# B&R Automation Studio project StructureSample
Automation Studio 4.12.8.41 SP

## Configuration Config1

CPU PC_any, AutomationRuntime Q4.93, Build 4.1.2, Vc V4.73.3

### Task classes (Cpu.sw)
```
Cyclic#8 (cycle 50000 us):
  StructureT <- GetVarStructure.prg
Binaries: udbdef, FWRules, TCData, iomap, ashwac, Role, sysconf, arconfig, asfw, User, ashwd
Libraries: AsBrStr, sys_lib, ArEventLog, runtime, AdvIecChk
```

### Hardware
```
PC : PC_any v1.1.1.0 (OrderNumber=PC)
  ConfigurationID = StructureTest_Config1
  Cyclic8Duration = 50000
  FileDevice1
  FileDeviceName1 = USER
  FileDevicePath1 = USER_PATH
```

## Logical view

Binary libraries used (declarations not repeated): operator, runtime, astime, AsIecCon, AsBrStr, sys_lib, ArEventLog

### Global.typ - Global data types
```iecst
TYPE
	testEnum :
		(
		red,
		green
		);
	testStructure : 	STRUCT
		Var1 : USINT;
		Var2 : UDINT;
		Var3 : ARRAY[0..5]OF UDINT;
		Enum : testEnum;
		RealLongVariableName : testSubStructure;
		SubStructure : testSubSubStructure;
	END_STRUCT;
	testSubStructure : 	STRUCT
		Var1234567 : STRING[80];
		Var22 : UDINT;
		EvenLongerSubVariableName : testSubSubStructure;
	END_STRUCT;
	testSubSubStructure : 	STRUCT
		Var11 : STRING[80];
		Var22 : UDINT;
		TheLongestSubVariableNameInisde : ARRAY[0..5]OF USINT;
	END_STRUCT;
END_TYPE
```

### Global.var - Global variables
```iecst
VAR
	testvariable_org : testStructure;
	testvariable_cpy : testStructure;
END_VAR
```

### Package Logical/Libraries - Global libraries

### Library Logical/Libraries/AdvIecChk (IEC, version 2.00.0) - IEC Check w/ Advanced Debugging Data
Depends on: Sys_Lib, AsBrStr, ArEventLog

#### AdvIecChk.fun - Exported functions and function blocks
```iecst
(************************************************************************************

Advanced IEC Check Functions Library

File: AdvIecChk.fun
Description: Declaration of library functions

!! Note: See the Automation Studio Help file before modifying these declarations!   !!
!! Most of these functions must be declared exactly as-is in order for the          !!
!! processor to recognize them as check functions. The implementation can change    !!
!! but the declaration cannot!                                                      !!

Authors:
    - Matt Adams (B&R Industrial Automation)
    - Varad Darji (B&R Industrial Automation)
    - Marcus Mangel (B&R Industrial Automation)

************************************************************************************)

FUNCTION CheckDivSint : SINT (*Called before the division/module using a SINT value. Returns the divisor if no errors are found*)
	VAR_INPUT
		divisor : SINT; (*For division: Value that should be divided by. For modulo: Right operand*)
	END_VAR
END_FUNCTION

FUNCTION CheckDivUsint : USINT (*Called before the division/module using a USINT value. Returns the divisor if no errors are found*)
	VAR_INPUT
		divisor : USINT; (*For division: Value that should be divided by. For modulo: Right operand*)
	END_VAR
END_FUNCTION

FUNCTION CheckDivInt : INT (*Called before the division/module using a INT value. Returns the divisor if no errors are found*)
	VAR_INPUT
		divisor : INT; (*For division: Value that should be divided by. For modulo: Right operand*)
	END_VAR
END_FUNCTION

FUNCTION CheckDivUint : UINT (*Called before the division/module using a UINT value. Returns the divisor if no errors are found*)
	VAR_INPUT
		divisor : UINT; (*For division: Value that should be divided by. For modulo: Right operand*)
	END_VAR
END_FUNCTION

FUNCTION CheckDivDint : DINT (*Called before the division/module using a DINT value. Returns the divisor if no errors are found*)
	VAR_INPUT
		divisor : DINT; (*For division: Value that should be divided by. For modulo: Right operand*)
	END_VAR
END_FUNCTION

FUNCTION CheckDivUdint : UDINT (*Called before the division/module using a UDINT value. Returns the divisor if no errors are found*)
	VAR_INPUT
		divisor : UDINT; (*For division: Value that should be divided by. For modulo: Right operand*)
	END_VAR
END_FUNCTION

FUNCTION CheckDivReal : REAL (*Called before the division/module using a REAL value. Returns the divisor if no errors are found*)
	VAR_INPUT
		divisor : REAL; (*For division: Value that should be divided by. For modulo: Right operand*)
	END_VAR
END_FUNCTION

FUNCTION CheckDivLReal : LREAL (*Called before the division/module using a LREAL value. Returns the divisor if no errors are found. (Cannot be used on SG3 or SGC targets)*)
	VAR_INPUT
		divisor : LREAL; (*For division: Value that should be divided by. For modulo: Right operand*)
	END_VAR
END_FUNCTION

FUNCTION CheckBounds : DINT (*Called before accessing an array. Returns the index if no errors are found. Otherwise, returns the problematic index bound*)
	VAR_INPUT
		index : DINT; (*Index being accessed*)
		lower : DINT; (*Lower bound (lowest possible index) of the array*)
		upper : DINT; (*Upper bound (highest possible index) of the array*)
	END_VAR
	VAR
		LowString : STRING[ADVIECCHK_MAX_STRING_LEN]; (*[INTERNAL] Lower bound as a string*)
		UpString : STRING[ADVIECCHK_MAX_STRING_LEN]; (*[INTERNAL] Upper bound as a string*)
		IndexString : STRING[ADVIECCHK_MAX_STRING_LEN]; (*[INTERNAL] Index as a string*)
		ErrorText : STRING[ADVIECCHK_MAX_STRING_LEN]; (*[INTERNAL] Error text created for a long entry based on input data*)
	END_VAR
END_FUNCTION

FUNCTION CheckRange : DINT (*Called before write accessing an enumeration variable. Returns the value if no errors are found. Otherwise, returns the problematic value bound*)
	VAR_INPUT
		value : DINT; (*Enumeration value being accessed*)
		lower : DINT; (*Lower bound (lowest possible value) of the enumeration*)
		upper : DINT; (*Upper bound (highest possible value) of the enumeration*)
	END_VAR
	VAR
		LowString : STRING[ADVIECCHK_MAX_STRING_LEN]; (*[INTERNAL] Lower bound as a string*)
		UpString : STRING[ADVIECCHK_MAX_STRING_LEN]; (*[INTERNAL] Upper bound as a string*)
		ValueString : STRING[ADVIECCHK_MAX_STRING_LEN]; (*[INTERNAL] Value as a string*)
		ErrorText : STRING[ADVIECCHK_MAX_STRING_LEN]; (*[INTERNAL] Error text created for a long entry based on input data*)
	END_VAR
END_FUNCTION

FUNCTION CheckSignedSubrange : DINT (*Called before write access to a variable with the data type "Subrange" if the subrange is used on a signed data type. Returns the value if no errors are found.
Otherwise, returns the problematic value bound*)
	VAR_INPUT
		value : DINT; (*Index being accessed*)
		lower : DINT; (*Lower bound (lowest possible index) of the subrange*)
		upper : DINT; (*Upper bound (highest possible index) of the subrange*)
	END_VAR
	VAR
		LowString : STRING[ADVIECCHK_MAX_STRING_LEN]; (*[INTERNAL] Lower bound as a string*)
		UpString : STRING[ADVIECCHK_MAX_STRING_LEN]; (*[INTERNAL] Lower bound as a string*)
		ValueString : STRING[ADVIECCHK_MAX_STRING_LEN]; (*[INTERNAL] Value as a string*)
		ErrorText : STRING[ADVIECCHK_MAX_STRING_LEN]; (*[INTERNAL] Error text created for a long entry based on input data*)
	END_VAR
END_FUNCTION

FUNCTION CheckUnsignedSubrange : UDINT (*Called before write access to a variable with the data type "Subrange" if the subrange is used on an unsigned data type. Returns the value if no errors are found.
Otherwise, returns the problematic value bound*)
	VAR_INPUT
		value : UDINT; (*Index being accessed*)
		lower : UDINT; (*Lower bound (lowest possible index) of the subrange*)
		upper : UDINT; (*Upper bound (highest possible index) of the subrange*)
	END_VAR
	VAR
		LowString : STRING[ADVIECCHK_MAX_STRING_LEN]; (*[INTERNAL] Lower bound as a string*)
		UpString : STRING[ADVIECCHK_MAX_STRING_LEN]; (*[INTERNAL] Upper bound as a string*)
		ValueString : STRING[ADVIECCHK_MAX_STRING_LEN]; (*[INTERNAL] Value as a string*)
		ErrorText : STRING[ADVIECCHK_MAX_STRING_LEN]; (*[INTERNAL] Error text created for a long entry based on input data*)
	END_VAR
END_FUNCTION

FUNCTION CheckReadAccess : UDINT (*Called before (read) accessing a memory address using a dynamic variable (ADR). Returns the input address*)
	VAR_INPUT
		address : UDINT; (*Address of the memory area being accessed*)
	END_VAR
END_FUNCTION

FUNCTION CheckWriteAccess : UDINT (*Called before (write) accessing a memory address using a dynamic variable (ADR). Returns the input address*)
	VAR_INPUT
		address : UDINT; (*Address of the memory area being accessed*)
	END_VAR
END_FUNCTION

FUNCTION MakeEntry : UDINT (*Creates a Logger entry detailing any errors. Returns a pointer to out_text*)
	VAR_INPUT
		ErrorCode : UINT; (*Error code that is used to generate a logbook Entry ID. Valid values are 0 to 65535*)
		ErrorText : STRING[ADVIECCHK_MAX_STRING_LEN]; (*Message string for the logbook. Additional characters will be added by the function before publishing the logbook entry*)
	END_VAR
	VAR
		taskname : STRING[ADVIECCHK_MAX_STRING_LEN]; (*[INTERNAL] Name of the task which caused the error. From ST_name()*)
		group : USINT; (*[INTERNAL] Task group number - See docs for ST_name in sys_lib. This will always be zero*)
		status_name : UINT; (*[INTERNAL] Return status of ST_name()*)
		out_text : STRING[ADVIECCHK_MAX_STRING_LEN]; (*[INTERNAL] Final error message text that is written to the logbook. Must be null terminated and maximum 32 characters (see ERRxwarning() docs)*)
		error_facility : UINT; (*[INTERNAL] Facility used to create the log Event ID. See ArEventLog documentation*)
		fb_ArEventLogGetIdent : ArEventLogGetIdent; (*[INTERNAL] Function block to get the ident of a logbook*)
		fb_ArEventLogWrite : ArEventLogWrite; (*[INTERNAL] Function block to write a log entry to the logbook*)
	END_VAR
END_FUNCTION

FUNCTION StrCatToMaxLen : UDINT (*Concatenates two strings, but keeps the result under the max allowed length. Also ensures the the string ends in a zero (null). Returns the length of the new string*)
	VAR_INPUT
		pDest : UDINT; (*Address of the destination string (will be modified)*)
		pSrc : UDINT; (*Address of the source string (not modified)*)
		MaxLength : UDINT; (*Maximum character length of the destination string*)
	END_VAR
	VAR
		destLen : UDINT; (*[INTERNAL] Holds the length of the string at pDest*)
		srcLen : UDINT; (*[INTERNAL] Holds the length of the string at pSrc*)
		lenToCopy : UDINT; (*[INTERNAL] Number of bytes to be copied, in the case of a partial string*)
	END_VAR
END_FUNCTION
```

#### AdvIecChk.st - Implementation file
```iecst
(************************************************************************************

Advanced IEC Check Functions Library

File: AdvIecChk.st
Description: Implentation of library functions
Authors:
    - Matt Adams (B&R Industrial Automation)
    - Varad Darji (B&R Industrial Automation)
    - Marcus Mangel (B&R Industrial Automation)

************************************************************************************)

(* Called before the division/module using a SINT value. Returns the divisor if no errors are found *)
(* Replaces CheckDivByte, which may return incorrect results *)
FUNCTION CheckDivSint

    IF divisor=0 THEN
        CheckDivSint := 1;
        MakeEntry(55555,'SINT division by 0');
    ELSE
        CheckDivSint := divisor;
    END_IF

END_FUNCTION

(* Called before the division/module using a USINT value. Returns the divisor if no errors are found *)
(* Replaces CheckDivByte, which may return incorrect results *)
FUNCTION CheckDivUsint

    IF divisor=0 THEN
        CheckDivUsint := 1;
        MakeEntry(55555,'USINT division by 0');
    ELSE
        CheckDivUsint := divisor;
    END_IF

END_FUNCTION

(* Called before the division/module using an INT value. Returns the divisor if no errors are found *)
(* Replaces CheckDivWord, which may return incorrect results *)
FUNCTION CheckDivInt

    IF divisor=0 THEN
        CheckDivInt := 1;
        MakeEntry(55555,'INT division by 0');
    ELSE
        CheckDivInt := divisor;
    END_IF

END_FUNCTION

(* Called before the division/module using a UINT value. Returns the divisor if no errors are found *)
(* Replaces CheckDivWord, which may return incorrect results *)
FUNCTION CheckDivUint

    IF divisor=0 THEN
        CheckDivUint := 1;
        MakeEntry(55555,'UINT division by 0');
    ELSE
        CheckDivUint := divisor;
    END_IF

END_FUNCTION

(* Called before the division/module using a DINT value. Returns the divisor if no errors are found *)
(* Replaces CheckDivDWord, which may return incorrect results *)
FUNCTION CheckDivDint

    IF divisor=0 THEN
        CheckDivDint := 1;
        MakeEntry(55555,'DINT division by 0');
    ELSE
        CheckDivDint := divisor;
    END_IF

END_FUNCTION

(* Called before the division/module using a UDINT value. Returns the divisor if no errors are found *)
(* Replaces CheckDivDWord, which may return incorrect results *)
FUNCTION CheckDivUdint

    IF divisor=0 THEN
        CheckDivUdint := 1;
        MakeEntry(55555,'UDINT division by 0');
    ELSE
        CheckDivUdint := divisor;
    END_IF

END_FUNCTION

(* Called before the division/module using a REAL value. Returns the divisor if no errors are found *)
FUNCTION CheckDivReal

    IF divisor=0 THEN
        CheckDivReal := 1;
        MakeEntry(55555,'REAL division by 0');
    ELSE
        CheckDivReal := divisor;
    END_IF

END_FUNCTION

(* Called before the division/module using a LREAL value. Returns the divisor if no errors are found *)
(* CANNOT BE USED on SG3 OR SGC targets!! *)
FUNCTION CheckDivLReal

    IF divisor=0 THEN
        CheckDivLReal := 1;
        MakeEntry(55555,'LREAL division by 0');
    ELSE
        CheckDivLReal := divisor;
    END_IF

END_FUNCTION

(* Called before accessing an array. Returns the index if no errors are found.
Otherwise, returns the problematic index bound *)
FUNCTION CheckBounds

    IF index < lower THEN
        CheckBounds := lower; // Unless: See end of function
        brsitoa(lower, ADR(LowString));
        brsitoa(upper, ADR(UpString));
        brsitoa(index, ADR(IndexString));
        brsstrcpy(ADR(ErrorText),ADR('Array Index '));
        StrCatToMaxLen(ADR(ErrorText),ADR(IndexString),ADVIECCHK_MAX_STRING_LEN);
        StrCatToMaxLen(ADR(ErrorText),ADR(' is outside range ['),ADVIECCHK_MAX_STRING_LEN);
        StrCatToMaxLen(ADR(ErrorText),ADR(LowString),ADVIECCHK_MAX_STRING_LEN);
        StrCatToMaxLen(ADR(ErrorText),ADR('..'),ADVIECCHK_MAX_STRING_LEN);
        StrCatToMaxLen(ADR(ErrorText),ADR(UpString),ADVIECCHK_MAX_STRING_LEN);
        StrCatToMaxLen(ADR(ErrorText),ADR(']'),ADVIECCHK_MAX_STRING_LEN);
        MakeEntry(55555,ErrorText);
    ELSIF index > upper THEN
        CheckBounds := upper; // Unless: See end of function
        brsitoa(lower, ADR(LowString));
        brsitoa(upper, ADR(UpString));
        brsitoa(index, ADR(IndexString));
        brsstrcpy(ADR(ErrorText),ADR('Array Index '));
        StrCatToMaxLen(ADR(ErrorText),ADR(IndexString),ADVIECCHK_MAX_STRING_LEN);
        StrCatToMaxLen(ADR(ErrorText),ADR(' is outside range ['),ADVIECCHK_MAX_STRING_LEN);
        StrCatToMaxLen(ADR(ErrorText),ADR(LowString),ADVIECCHK_MAX_STRING_LEN);
        StrCatToMaxLen(ADR(ErrorText),ADR('..'),ADVIECCHK_MAX_STRING_LEN);
        StrCatToMaxLen(ADR(ErrorText),ADR(UpString),ADVIECCHK_MAX_STRING_LEN);
        StrCatToMaxLen(ADR(ErrorText),ADR(']'),ADVIECCHK_MAX_STRING_LEN);
        MakeEntry(55555,ErrorText);
    ELSE
        CheckBounds := index;
    END_IF

END_FUNCTION

(* Called before write accessing an enumeration variable. Returns the value if no errors are found.
Otherwise, returns the problematic value bound *)
FUNCTION CheckRange

	IF value < lower THEN
		CheckRange := lower; // Unless: See end of function
		brsitoa(lower, ADR(LowString));
		brsitoa(upper, ADR(UpString));
		brsitoa(value, ADR(ValueString));
		brsstrcpy(ADR(ErrorText),ADR('Enumeration Value '));
		StrCatToMaxLen(ADR(ErrorText),ADR(ValueString),ADVIECCHK_MAX_STRING_LEN);
		StrCatToMaxLen(ADR(ErrorText),ADR(' is outside range ['),ADVIECCHK_MAX_STRING_LEN);
		StrCatToMaxLen(ADR(ErrorText),ADR(LowString),ADVIECCHK_MAX_STRING_LEN);
		StrCatToMaxLen(ADR(ErrorText),ADR('..'),ADVIECCHK_MAX_STRING_LEN);
		StrCatToMaxLen(ADR(ErrorText),ADR(UpString),ADVIECCHK_MAX_STRING_LEN);
		StrCatToMaxLen(ADR(ErrorText),ADR(']'),ADVIECCHK_MAX_STRING_LEN);
		MakeEntry(55555,ErrorText);
	ELSIF value > upper THEN
		CheckRange := upper; // Unless: See end of function
		brsitoa(lower, ADR(LowString));
		brsitoa(upper, ADR(UpString));
		brsitoa(value, ADR(ValueString));
		brsstrcpy(ADR(ErrorText),ADR('Enumeration Value '));
		StrCatToMaxLen(ADR(ErrorText),ADR(ValueString),ADVIECCHK_MAX_STRING_LEN);
		StrCatToMaxLen(ADR(ErrorText),ADR(' is outside range ['),ADVIECCHK_MAX_STRING_LEN);
		StrCatToMaxLen(ADR(ErrorText),ADR(LowString),ADVIECCHK_MAX_STRING_LEN);
		StrCatToMaxLen(ADR(ErrorText),ADR('..'),ADVIECCHK_MAX_STRING_LEN);
		StrCatToMaxLen(ADR(ErrorText),ADR(UpString),ADVIECCHK_MAX_STRING_LEN);
		StrCatToMaxLen(ADR(ErrorText),ADR(']'),ADVIECCHK_MAX_STRING_LEN);
		MakeEntry(55555,ErrorText);
	ELSE
		CheckRange := value;
	END_IF

END_FUNCTION

(* Called before write access to a variable with the data type "Subrange" if the subrange is used on a signed data type. Returns the value if no errors are found.
Otherwise, returns the problematic value bound *)
FUNCTION CheckSignedSubrange

    IF value < lower THEN
        CheckSignedSubrange := lower; // Unless: See end of function
        brsitoa(lower, ADR(LowString));
        brsitoa(upper, ADR(UpString));
        brsitoa(value, ADR(ValueString));
        brsstrcpy(ADR(ErrorText),ADR('Signed Subrange Index '));
        StrCatToMaxLen(ADR(ErrorText),ADR(ValueString),ADVIECCHK_MAX_STRING_LEN);
        StrCatToMaxLen(ADR(ErrorText),ADR(' is outside range ['),ADVIECCHK_MAX_STRING_LEN);
        StrCatToMaxLen(ADR(ErrorText),ADR(LowString),ADVIECCHK_MAX_STRING_LEN);
        StrCatToMaxLen(ADR(ErrorText),ADR('..'),ADVIECCHK_MAX_STRING_LEN);
        StrCatToMaxLen(ADR(ErrorText),ADR(UpString),ADVIECCHK_MAX_STRING_LEN);
        StrCatToMaxLen(ADR(ErrorText),ADR(']'),ADVIECCHK_MAX_STRING_LEN);
        MakeEntry(55555,ErrorText);
    ELSIF value > upper THEN
        CheckSignedSubrange := upper; // Unless: See end of function
        brsitoa(lower, ADR(LowString));
        brsitoa(upper, ADR(UpString));
        brsitoa(value, ADR(ValueString));
        StrCatToMaxLen(ADR(ErrorText),ADR('Signed Subrange Index '),ADVIECCHK_MAX_STRING_LEN);
        StrCatToMaxLen(ADR(ErrorText),ADR(ValueString),ADVIECCHK_MAX_STRING_LEN);
        StrCatToMaxLen(ADR(ErrorText),ADR(' is outside range ['),ADVIECCHK_MAX_STRING_LEN);
        StrCatToMaxLen(ADR(ErrorText),ADR(LowString),ADVIECCHK_MAX_STRING_LEN);
        StrCatToMaxLen(ADR(ErrorText),ADR('..'),ADVIECCHK_MAX_STRING_LEN);
        StrCatToMaxLen(ADR(ErrorText),ADR(UpString),ADVIECCHK_MAX_STRING_LEN);
        StrCatToMaxLen(ADR(ErrorText),ADR(']'),ADVIECCHK_MAX_STRING_LEN);
        MakeEntry(55555,ErrorText);
    ELSE
        CheckSignedSubrange := value;
    END_IF

END_FUNCTION

(* Called before write access to a variable with the data type "Subrange" if the subrange is used on an unsigned data type. Returns the value if no errors are found.
Otherwise, returns the problematic value bound *)
FUNCTION CheckUnsignedSubrange

    IF value < lower THEN
        CheckUnsignedSubrange := lower; // Unless: See end of function
        brsitoa(lower, ADR(LowString));
        brsitoa(upper, ADR(UpString));
        brsitoa(value, ADR(ValueString));
        brsstrcpy(ADR(ErrorText),ADR('Unsigned Subrange Index '));
        StrCatToMaxLen(ADR(ErrorText),ADR(ValueString),ADVIECCHK_MAX_STRING_LEN);
        StrCatToMaxLen(ADR(ErrorText),ADR(' is outside range ['),ADVIECCHK_MAX_STRING_LEN);
        StrCatToMaxLen(ADR(ErrorText),ADR(LowString),ADVIECCHK_MAX_STRING_LEN);
        StrCatToMaxLen(ADR(ErrorText),ADR('..'),ADVIECCHK_MAX_STRING_LEN);
        StrCatToMaxLen(ADR(ErrorText),ADR(UpString),ADVIECCHK_MAX_STRING_LEN);
        StrCatToMaxLen(ADR(ErrorText),ADR(']'),ADVIECCHK_MAX_STRING_LEN);
        MakeEntry(55555,ErrorText);
    ELSIF value > upper THEN
        CheckUnsignedSubrange := upper; // Unless: See end of function
        brsitoa(lower, ADR(LowString));
        brsitoa(upper, ADR(UpString));
        brsitoa(value, ADR(ValueString));
        brsstrcpy(ADR(ErrorText),ADR('Unsigned Subrange Index '));
        StrCatToMaxLen(ADR(ErrorText),ADR(ValueString),ADVIECCHK_MAX_STRING_LEN);
        StrCatToMaxLen(ADR(ErrorText),ADR(' is outside range ['),ADVIECCHK_MAX_STRING_LEN);
        StrCatToMaxLen(ADR(ErrorText),ADR(LowString),ADVIECCHK_MAX_STRING_LEN);
        StrCatToMaxLen(ADR(ErrorText),ADR('..'),ADVIECCHK_MAX_STRING_LEN);
        StrCatToMaxLen(ADR(ErrorText),ADR(UpString),ADVIECCHK_MAX_STRING_LEN);
        StrCatToMaxLen(ADR(ErrorText),ADR(']'),ADVIECCHK_MAX_STRING_LEN);
        MakeEntry(55555,ErrorText);
    ELSE
        CheckUnsignedSubrange := value;
    END_IF

END_FUNCTION

(* Called before (read) accessing a memory address using a dynamic variable (ADR). Returns the input address *)
// Note: We cannot substitute in any addresses here
// This always returns a zero address
// That means a pagefault will occur no matter what, but at least we can log why
FUNCTION CheckReadAccess

    IF address=0 THEN
        MakeEntry(55555,'Read from memory address of zero');
        CheckReadAccess:=0;
    ELSE
        CheckReadAccess:=address;
    END_IF

END_FUNCTION

(* Called before (write) accessing a memory address using a dynamic variable (ADR). Returns the input address *)
// Note: We cannot substitute in any addresses here
// This always returns a zero address
// That means a pagefault will occur no matter what, but at least we can log why
FUNCTION CheckWriteAccess

    IF address=0 THEN
        MakeEntry(55555,'Write to memory address of zero');
        CheckWriteAccess:=0;
    ELSE
        CheckWriteAccess:=address;
    END_IF

END_FUNCTION

(* Creates a Logger entry detailing any errors. Returns a pointer to out_text *)
FUNCTION MakeEntry

    // Get task name and add to error text string
	status_name := ST_name(0,ADR(taskname),ADR(group));

	brsmemset(ADR(out_text),0,SIZEOF(out_text)); // We need to make sure the data is null terminated, so start with all zeros
	StrCatToMaxLen(ADR(out_text),ADR(ErrorText), ADVIECCHK_MAX_STRING_LEN);

	IF status_name = 0 THEN
		StrCatToMaxLen(ADR(out_text),ADR(' in task '), ADVIECCHK_MAX_STRING_LEN);
		StrCatToMaxLen(ADR(out_text),ADR('"'), ADVIECCHK_MAX_STRING_LEN);
		StrCatToMaxLen(ADR(out_text),ADR(taskname), ADVIECCHK_MAX_STRING_LEN);
		StrCatToMaxLen(ADR(out_text),ADR('"'), ADVIECCHK_MAX_STRING_LEN);
	END_IF;

	// Finalize logbook entry - Write to the existing User logbook
	// It would be possible to create our own logbook, but that would be much more complex
	error_facility := 0; // See ArEventLog documentation on the 32-bit event ID

	fb_ArEventLogGetIdent.Execute := TRUE;
	fb_ArEventLogGetIdent.Name := '$$arlogusr'; // This is the only system logbook we can access
	fb_ArEventLogGetIdent();

	fb_ArEventLogWrite.Execute := TRUE;
	fb_ArEventLogWrite.Ident := fb_ArEventLogGetIdent.Ident;
	fb_ArEventLogWrite.EventID := ArEventLogMakeEventID(arEVENTLOG_SEVERITY_ERROR,error_facility,ErrorCode);
	fb_ArEventLogWrite.AddData := ADR(out_text);
	fb_ArEventLogWrite.AddDataFormat := arEVENTLOG_ADDFORMAT_TEXT;
	fb_ArEventLogWrite.AddDataSize := MIN(SIZEOF(out_text),brsstrlen(ADR(out_text))+1); // If string doesn't fill the whole buffer, take just it's length
	fb_ArEventLogWrite.ObjectID := 'AdvIecChk';                                         // plus the next char (should be a zero, this is the trailing null char)
	fb_ArEventLogWrite();

	MakeEntry := brsstrlen(ADR(out_text));

	brsmemcpy(1,1,1); // Create a pagefault on purpose to get the backtrace data

END_FUNCTION

(* Concatenates two strings, but keeps the result under the max allowed length.
Also ensures the the string ends in a zero (null).
Returns the length of the new string *)
FUNCTION StrCatToMaxLen

    IF (pDest = 0) OR (pSrc = 0) OR (MaxLength = 0) THEN
        StrCatToMaxLen := 0;
        RETURN;
    END_IF;

    destLen := brsstrlen(pDest);
    srcLen := brsstrlen(pSrc);

    lenToCopy := MIN(srcLen,(MaxLength - destLen)); // Copy the full src string if possible, otherwise copy a partial string
    brsmemcpy(pDest + destLen, pSrc, lenToCopy);
    brsmemset(pDest + destLen + lenToCopy, 0, 1); // Ensure trailing null character
    StrCatToMaxLen := destLen + lenToCopy;

END_FUNCTION
```

#### AdvIecChk.var - Constant declarations
```iecst
(************************************************************************************

Advanced IEC Check Functions Library

File: AdvIecChk.var
Description: Constants used in the AdvIecChk library
Authors:
    - Marcus Mangel (B&R Industrial Automation)

************************************************************************************)
VAR CONSTANT
	ADVIECCHK_MAX_STRING_LEN : USINT := 64; (*Maximum character length for the error info string. Used to prevent buffer overflow*)
END_VAR
```

### Program Logical/GetVarStructure (IEC)

#### Main.st - Init, cyclic, exit code
```iecst
PROGRAM _INIT
	testvariable_org;
	testvariable_cpy;

END_PROGRAM

PROGRAM _CYCLIC
	// Call the structure loader functionblock to create a list of all members
	//StructureLoader_0.Enable := TRUE;
	StructureLoader_0.StructAdr := ADR('testvariable_org');
	StructureLoader_0();

	// This block compares the orginial structure against a backup
	// When a difference was detected the variable name is stored in 'diff_str'
	// The change can be acknowldged with 'ack'
	CASE compare OF
		1:
			// Call the structure loader functionblock to create a list of all members
			StructureLoader_1.Enable := TRUE;
			StructureLoader_1.StructAdr := ADR('testvariable_cpy');
			StructureLoader_1();

			IF StructureLoader_1.Done AND NOT StructureLoader_1.Error THEN
				i := 0;
				compare := 2;
			END_IF
		2:
			result := brsmemcmp(StructureLoader_1.StructDetails[i].Pointer, StructureLoader_0.StructDetails[i].Pointer, StructureLoader_1.StructDetails[i].DataLength);
			IF result <> 0 THEN
				diff_str := StructureLoader_0.StructDetails[i].Name;
				compare := 3;
			ELSIF i < StructureLoader_0.StructEntries THEN
				i := i + 1;
			ELSE
				i := 0;
			END_IF
		3:
			IF ack THEN
				brsmemcpy(StructureLoader_1.StructDetails[i].Pointer, StructureLoader_0.StructDetails[i].Pointer, StructureLoader_1.StructDetails[i].DataLength);
				i := 0;
				ack := 0;
				diff_str := '';
				compare := 2;
			END_IF

	END_CASE;

END_PROGRAM
```

#### Variables.var - Local variables
```iecst
(*Load structure details*)
VAR
	StructureLoader_0 : StructureLoader := (0);
END_VAR
(*Compare structures*)
VAR
	StructureLoader_1 : StructureLoader := (0); (*Second instance for backup structure*)
	compare : USINT; (*Start compare with 1*)
	i : UINT;
	result : UDINT;
	diff_str : STRING[MAX_VARIABLE_NAME_LEN]; (*String containing the variable name where a difference was detected*)
	ack : BOOL; (*Acknowledge the change*)
END_VAR
```

#### StructFunctions.fun
```iecst
FUNCTION_BLOCK StructureLoader
	VAR_INPUT
		Enable : BOOL; (*Will recursively load the structure and all structures inside the structure who's variable name is provided via StructAdr*)
		StructAdr : REFERENCE TO STRING[200]; (*Pointer to a string of the structure to be loaded*)
	END_VAR
	VAR_OUTPUT
		Busy : BOOL;
		Done : BOOL;
		Error : BOOL;
		ErrorText : STRING[200];
		ErrorCode : UINT;
		StructSize : UDINT;
		StructEntries : UINT;
		StructDetails : ARRAY[0..MAX_VARIABLE_IDX] OF StructLoad_Data_TYP;
	END_VAR
	VAR
		Internal : StructInternal_TYP;
		zzEdge00000 : BOOL;
		zzEdge00001 : BOOL;
	END_VAR
END_FUNCTION_BLOCK
```

#### StructTypes.typ - Local data types
```iecst
TYPE
	StructLoad_Data_TYP : 	STRUCT
		Name : STRING[MAX_VARIABLE_NAME_LEN]; (*Member's name*)
		Pointer : UDINT; (*Member's memory address*)
		Datatype : UDINT; (*Member's datatype (See ad7773ad-be51-4500-a7ba-b8f12743a77a for more info)*)
		DataLength : UDINT; (*Number of Byte the member memory consumes*)
		Dimension : UDINT; (*If an array, the number of array elements.  If a structure, the number of structure elements*)
	END_STRUCT;
	StructInternal_TYP : 	STRUCT
		StateMachine : StructData_StateMachine_TYP;
		StatusFunction : UINT;
		Index : UDINT;
		Cycles : UINT;
		DataList_Index : UINT;
		Structure_Index : ARRAY[0..MAX_STRUCT_DEPTH]OF USINT;
		SubStructure_Index : UDINT;
		Period_Index : UDINT;
		CurrentPath : STRING[TOTAL_STRUCTURE_NAME_LEN];
		CurrentSubPath : ARRAY[0..MAX_VARIABLE_NAME_LEN]OF USINT;
		CurrentMember : STRING[SINGLE_VARIABLE_NAME_LEN];
		CurrentPV : STRING[TOTAL_STRUCTURE_NAME_LEN];
		CurrentData : StructLoad_Data_TYP;
		tempIdxStr : STRING[10];
		tempNameStr : STRING[TOTAL_STRUCTURE_NAME_LEN];
		tempPointer : UDINT;
		tempDimension : UDINT; (*If an array, the number of array elements.  If a structure, the number of structure elements*)
	END_STRUCT;
	StructData_StateMachine_TYP :
		(
		STRUCTDATA_INIT, (*Initialize State !MUST BE FIRST!*)
		STRUCTDATA_WAIT_FOR_CMD, (*Function block will wait for a command in this state*)
		STRUCTDATA_LOAD, (*Loading is active*)
		STRUCTDATA_DONE, (*Loading is done*)
		STRUCTDATA_ERROR (*An error occured.  The error will be reset once the command is set low.*)
		);
END_TYPE
```

#### StructVariables.var - Local variables
```iecst
(*-------------------------------------------------------------------------------------------------------------------------------------------------------------------------------------------------------------------------------------------------------------------------------------------------------------------------------------------------*)
(*Change this according to your structure*)
VAR CONSTANT
	MAX_STRUCT_DEPTH : UINT := 10; (*Maximum depth of the structure*)
	MAX_VARIABLE_IDX : UINT := 100; (*Maximum number of variables in the structure, including all array indices*)
	MAX_VARIABLE_NAME_LEN : UINT := 200; (*Maximum length of a complete variable name*)
	OVERRIDE : UINT := 2; (*Number of executions per cycle*)
END_VAR
(*-------------------------------------------------------------------------------------------------------------------------------------------------------------------------------------------------------------------------------------------------------------------------------------------------------------------------------------------------*)
(*Dont change anything below this line*)
VAR CONSTANT
	SINGLE_VARIABLE_NAME_LEN : UINT := 33; (*Default length of variable. Dont change this value!*)
	TOTAL_STRUCTURE_NAME_LEN : UINT := SINGLE_VARIABLE_NAME_LEN+MAX_VARIABLE_NAME_LEN;
	ERR_VAR_TO_LONG : UINT := 10000; (*Total variable name is too long. Increase MAX_VARIABLE_NAME_LEN*)
	ERR_MAX_RECURSIONS : UINT := 10001; (*Max structure recursion exceeded. Increase MAX_STRUCT_DEPTH*)
	ERR_MAX_ENTRIES : UINT := 10002; (*Max number of enrties exceeded. Increase MAX_VARIABLE_IDX*)
END_VAR
```

#### StructureLoader.st
```iecst
FUNCTION_BLOCK StructureLoader

	IF EDGENEG(Enable) THEN
		Internal.StateMachine := STRUCTDATA_INIT;
	END_IF

	CASE (Internal.StateMachine) OF

		STRUCTDATA_INIT:
			// Clear Indexes and structures
			brsmemset(ADR(StructDetails), 0, SIZEOF(StructDetails));
			brsmemset(ADR(Internal), 0, SIZEOF(Internal));
			Error := FALSE;
			ErrorCode := 0;
			ErrorText := '';
			StructSize := 0;
			StructEntries := 0;
			Done := FALSE;

			Internal.StateMachine := STRUCTDATA_WAIT_FOR_CMD;

		STRUCTDATA_WAIT_FOR_CMD:

			IF EDGEPOS(Enable) THEN
				// Check if the pointer is good
				IF ADR(StructAdr) = 0 THEN
					Error := TRUE;
					ErrorText := 'PV name is NULL';
					Internal.StateMachine := STRUCTDATA_ERROR;
				ELSE
					Busy := TRUE;
					Done := FALSE;
					Internal.StateMachine := STRUCTDATA_LOAD;

				END_IF;
			END_IF;

		STRUCTDATA_LOAD:

			FOR Internal.Cycles:=0 TO OVERRIDE DO

				// Start with the main structure
				brsstrcpy(ADR(Internal.CurrentPath), ADR(StructAdr));
				brsstrcat(ADR(Internal.CurrentPath), ADR(Internal.CurrentSubPath));

				// Get basic variable information
				Internal.StatusFunction := PV_ninfo( ADR(StructAdr), ADR(Internal.CurrentData.Datatype), ADR(Internal.CurrentData.DataLength), ADR(Internal.CurrentData.Dimension));

				IF ErrorCode = 0 THEN
					StructSize := Internal.CurrentData.DataLength;
					GetStructureData;
					IF Internal.StateMachine <> STRUCTDATA_LOAD THEN
						EXIT;
					END_IF
				ELSE
					Error := TRUE;
					ErrorText := 'Failed to get struct size';
					Internal.StateMachine := STRUCTDATA_ERROR;
				END_IF;
			END_FOR;

		STRUCTDATA_DONE:

			Busy := FALSE;
			Done := TRUE;

			IF NOT Enable THEN
				Done := FALSE;
				Internal.StateMachine := STRUCTDATA_WAIT_FOR_CMD;
				StructEntries := 0;
			END_IF;

		STRUCTDATA_ERROR:
			ErrorCode := Internal.StatusFunction;

			IF NOT Enable THEN
				Error := FALSE;
				ErrorText := '';
				Internal.StateMachine := STRUCTDATA_WAIT_FOR_CMD;
			END_IF;

	END_CASE;

END_FUNCTION_BLOCK
```

#### StructureLoaderGetData.st
```iecst
ACTION GetStructureData:

	// Get the structure member
	Internal.StatusFunction := PV_item(ADR(Internal.CurrentPath), Internal.Structure_Index[Internal.SubStructure_Index], ADR(Internal.CurrentMember));

	IF Internal.StatusFunction = 0 THEN

		// Build complete members name
		IF Internal.SubStructure_Index > 0 THEN
			brsstrcpy(ADR(Internal.CurrentData.Name), ADR(Internal.CurrentSubPath[1]));

			// Make sure new name fits into destination
			IF brsstrlen(ADR(Internal.CurrentData.Name)) + brsstrlen(ADR(Internal.CurrentMember)) + 1 < SIZEOF(Internal.CurrentData.Name) THEN
				brsstrcat(ADR(Internal.CurrentData.Name), ADR('.') );
				brsstrcat(ADR(Internal.CurrentData.Name), ADR(Internal.CurrentMember));

			ELSE
				Error := TRUE;
				ErrorText := Internal.CurrentMember;
				brsstrcat(ADR(ErrorText), ADR(' <- excceeds the max length of MAX_VARIABLE_NAME_LEN'));
				Internal.StatusFunction := ERR_VAR_TO_LONG;
				Internal.StateMachine := STRUCTDATA_ERROR;
				RETURN;
			END_IF;
		ELSE

			Internal.CurrentData.Name := Internal.CurrentMember;
		END_IF;

		// Move variable full name
		brsstrcpy(ADR(Internal.CurrentPV), ADR(Internal.CurrentPath));

		// Make sure that new name fits into destination
		IF brsstrlen(ADR(Internal.CurrentPV)) + brsstrlen(ADR(Internal.CurrentMember)) + 1 < SIZEOF(Internal.CurrentPV) THEN
			brsstrcat(ADR(Internal.CurrentPV), ADR('.'));
			brsstrcat(ADR(Internal.CurrentPV), ADR(Internal.CurrentMember));

		ELSE

			Error := TRUE;
			ErrorText := Internal.CurrentMember;
			brsstrcat(ADR(ErrorText), ADR(' <- excceeds the max length of MAX_VARIABLE_NAME_LEN') );
			Internal.StatusFunction := ERR_VAR_TO_LONG;
			Internal.StateMachine := STRUCTDATA_ERROR;
			RETURN;
		END_IF;

		// Get variable details
		Internal.StatusFunction := PV_ninfo(ADR(Internal.CurrentPV), ADR(Internal.CurrentData.Datatype), ADR(Internal.CurrentData.DataLength), ADR(Internal.CurrentData.Dimension));

		IF Internal.StatusFunction = 0 THEN
			// Get the pointer to this variable
			Internal.StatusFunction := PV_xgetadr(ADR(Internal.CurrentPV), ADR(Internal.CurrentData.Pointer), ADR(Internal.CurrentData.DataLength));

			IF Internal.StatusFunction = 0 THEN

				// Check if the variable is a structure
				IF (Internal.CurrentData.Datatype = SYSLIB_IEC_TYPE_USER_DEFINED OR Internal.CurrentData.Datatype = SYSLIB_IEC_TYPE_USER_DEFINED_2) AND
					(Internal.CurrentData.DataLength <> 4) AND
					(Internal.CurrentData.Dimension <> 1) THEN

					// Move to the sub structure
					IF Internal.SubStructure_Index < MAX_STRUCT_DEPTH - 1 THEN
						//Add to the CurrentSubPath
						brsstrcat( ADR(Internal.CurrentSubPath), ADR('.') );
						brsstrcat( ADR(Internal.CurrentSubPath), ADR(Internal.CurrentMember) );

						//Move down a level in the structure
						Internal.SubStructure_Index := Internal.SubStructure_Index + 1;

						// Maximum number of recursion exceeded
					ELSE
						Error := TRUE;
						ErrorText := 'Max number of recursions exceeded, increase the value of MAX_STRUCT_DEPTH';
						Internal.StatusFunction := ERR_MAX_RECURSIONS;
						Internal.StateMachine := STRUCTDATA_ERROR;
					END_IF;

					// Variable is not a structure
				ELSE

					AddData;
				END_IF;
			ELSE

				Error := TRUE;
				ErrorText := 'Failed to get pointer';
				Internal.StateMachine := STRUCTDATA_ERROR;
			END_IF;
		ELSE

			Error := TRUE;
			ErrorText := 'Failed to get variable details';
			Internal.StateMachine := STRUCTDATA_ERROR;
		END_IF;

		// 14704 - Invalid Component - This suggests that the index listed is not a member and the structure has ended
		// 14713 - No PV Description avalaible - This error is known to occur when requesting information about a variable that is not a structure (e.g. Could be an ENUM)
	ELSIF Internal.StatusFunction = 14704 OR Internal.StatusFunction = 14713 THEN

		// Check if this is the root structure
		IF Internal.SubStructure_Index = 0 THEN
			Busy := FALSE;
			Done := TRUE;
			StructEntries := Internal.DataList_Index;
			Internal.StateMachine := STRUCTDATA_DONE;

			// This is a sub-structure
		ELSE

			// Done searching the sub-structure, set the index to zero for next sub-structure
			Internal.Structure_Index[Internal.SubStructure_Index] := 0;

			// Move down a level in the structure tree
			Internal.SubStructure_Index := Internal.SubStructure_Index - 1;

			// Find the last period in the subpath, move down the structure tree, the path must move down a level as well
			Internal.Period_Index := 0;

			FOR Internal.Index := 0 TO SIZEOF(Internal.CurrentSubPath) - 1 DO
				IF (Internal.CurrentSubPath[Internal.Index] = 46 ) THEN
					Internal.Period_Index := Internal.Index;
				ELSIF (Internal.CurrentSubPath[Internal.Index] = 0 ) THEN
					EXIT;
				END_IF;
			END_FOR;

			//Erase the string up to the period
			Internal.CurrentSubPath[Internal.Period_Index] := 0;

			// Check if this is the end of structure or it is not a structure at all
			IF Internal.StatusFunction = 14704 THEN

				Internal.Structure_Index[Internal.SubStructure_Index] := Internal.Structure_Index[Internal.SubStructure_Index] + 1;
			ELSIF Internal.StatusFunction = 14713 THEN

				AddData;
			ELSE

				Error := TRUE;
				ErrorText := 'Unknown error';
				Internal.StateMachine := STRUCTDATA_ERROR;
			END_IF;

		END_IF;

	ELSE

		Error := TRUE;
		ErrorText := 'PV does not exist or not loaded';
		Internal.StateMachine := STRUCTDATA_ERROR;
	END_IF;

END_ACTION
```

#### StructureLoaderAddData.st
```iecst
ACTION AddData:

	// Make sure that we dont exceed the maximum list of entries
	IF Internal.DataList_Index < SIZEOF(StructDetails)/SIZEOF(StructDetails[0]) THEN

		// Add each array element to the list
		IF Internal.CurrentData.Dimension > 1 THEN

			// Save the name of the base variable
			Internal.tempNameStr := Internal.CurrentData.Name;
			Internal.tempPointer := Internal.CurrentData.Pointer;

			// Get details for first element
			brsstrcat(ADR(Internal.CurrentPV), ADR('[0]'));
			Internal.StatusFunction := PV_ninfo(ADR(Internal.CurrentPV), ADR(Internal.CurrentData.Datatype), ADR(Internal.CurrentData.DataLength), ADR(Internal.tempDimension));

			IF Internal.StatusFunction = 0 THEN

				FOR Internal.Index := 0 TO Internal.CurrentData.Dimension - 1 DO
					// Refresh the base variable name
					Internal.CurrentData.Name := Internal.tempNameStr;

					// Append the array index, starting at 0
					brsstrcat(ADR(Internal.CurrentData.Name), ADR('['));
					brsitoa(Internal.Index, ADR(Internal.tempIdxStr));
					brsstrcat(ADR(Internal.CurrentData.Name), ADR(Internal.tempIdxStr));
					brsstrcat(ADR(Internal.CurrentData.Name), ADR(']'));

					// Shift pointer based on Datalength of the pointed to variable
					Internal.CurrentData.Pointer := Internal.tempPointer + (DINT_TO_UDINT(Internal.Index) * Internal.CurrentData.DataLength);

					// Check if the current index in the data list is lower than the size of the data list
					IF Internal.DataList_Index < SIZEOF(StructDetails)/SIZEOF(StructDetails[0]) THEN

						// Move the data into the final output structure
						brsmemcpy(ADR(StructDetails[Internal.DataList_Index]), ADR(Internal.CurrentData), SIZEOF(StructDetails[0]));
					ELSE

						Error := TRUE;
						ErrorText := 'No more entries available, increase the value of MAX_VARIABLE_IDX';
						Internal.StatusFunction := ERR_MAX_ENTRIES;
						Internal.StateMachine := STRUCTDATA_ERROR;
						RETURN;
					END_IF

					// Goto the next data list member
					Internal.DataList_Index := Internal.DataList_Index + 1;

				END_FOR

			ELSE

				Error := TRUE;
				ErrorText := 'Failed to get variable details';
				Internal.StateMachine := STRUCTDATA_ERROR;
			END_IF;

		ELSE

			// Move the data into the final output structure
			brsmemcpy(ADR(StructDetails[Internal.DataList_Index]), ADR(Internal.CurrentData), SIZEOF(StructDetails[0]));

			// Goto the next data list member
			Internal.DataList_Index := Internal.DataList_Index + 1;

		END_IF

		// Goto the next member index in the current stuctured directory
		Internal.Structure_Index[Internal.SubStructure_Index] := Internal.Structure_Index[Internal.SubStructure_Index] + 1;

	ELSE

		Error := TRUE;
		ErrorText := 'No more entries available. Increase the value of MAX_VARIABLE_IDX';
		Internal.StateMachine := STRUCTDATA_ERROR;
	END_IF;

END_ACTION
```
